FUNCTION_BLOCK FB_ModbusSlaveTcp EXTENDS FB_UniversalModbusSlave IMPLEMENTS I_ModbusSlaveTcp
VAR
	sIPAddr       : STRING(15);
	nTCPPort	  : UINT:= 502;//MODBUS_TCP_PORT
	nErrId     	  : UDINT;
END_VAR

PROPERTY IpAddr : String(15)
GET
IpAddr := sIPAddr;
END_GET
SET
sIPAddr := IpAddr;
END_SET
END_PROPERTY

PROPERTY ModbusErrorID : UDINT
GET
ModbusErrorID := nErrId;
END_GET
SET
nErrId := ModbusErrorID;
END_SET
END_PROPERTY

PROPERTY TcpPort : Uint
GET
TcpPort := nTCPPort;
END_GET
SET
nTCPPort := TcpPort;
END_SET
END_PROPERTY

END_FUNCTION_BLOCK

(* stored: Version 1.1.0.1, ProductVersion 3.1.4024.12
   POU FB_ModbusSlaveTcp: Id {37164e8e-1317-4a02-a421-ddb976abba2c}, SpecialFunc None
   Property IpAddr: Id {c6680cec-1927-4f98-970b-41887a193eb1}
   Get Get: Id {136072bd-17ff-4cf1-93f2-df162ca9d629}
   Set Set: Id {0cd7b8ba-b2d7-4e13-a558-8d8f869f35d8}
   Property ModbusErrorID: Id {e82491a5-78ab-4ab5-9793-d32aea28c506}
   Get Get: Id {80cc5a48-f84c-4f4b-a462-9390916f9cb6}
   Set Set: Id {ce6d558a-d8e8-435f-8fe2-6145a6b43c53}
   Property TcpPort: Id {44a0460a-3f7c-492f-bcb8-3da62b5eaf28}
   Get Get: Id {e70408a0-588f-4095-8ca2-a7a2032008ba}
   Set Set: Id {477b12b6-7881-4ccb-b167-4acafe840d79} *)
